FUNCTION_BLOCK FB_TP_LTIME (* standard timer function block (pulse) (LTIME) *)
  (* Standard: 61131-3; Classification: standard timer function block; Description: Copyright (c) 2011 TU Wien ACIN, Patrick Aigner, HR Agrartechnik GmbH This program and the accompanying materials are made available under the terms of the Eclipse Public License 2.0 which is available at https://www.eclipse.org/legal/epl-2.0/ SPDX-License-Identifier: EPL-2.0 Some portions generated by Gemini CLI *)
  (* Version 1.0, 2026-02-01, Franz Höpfinger, HR Agrartechnik GmbH, Copy over from FB_TP and made this Block *)
  PACKAGE iec61131::timers;
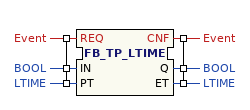
  EVENT_INPUT
    REQ WITH IN, PT; (* Service Request *)
  END_EVENT
  EVENT_OUTPUT
    CNF WITH Q, ET; (* Confirmation of Requested Service *)
  END_EVENT
  VAR_INPUT
    IN : BOOL; (* Input *)
    PT : LTIME; (* Pulse time *)
  END_VAR
  VAR_OUTPUT
    Q : BOOL; (* output *)
    ET : LTIME; (* elapse time *)
  END_VAR
  VAR
    MEM : BOOL; (* internal variable *)
    StartTime : LTIME; (* internal variable *)
  END_VAR
  EC_STATES
    REQ : REQ -> CNF;
  END_STATES
  ALGORITHM REQ IN ST:
VAR_TEMP
	SysTime : TIME;
END_VAR

SysTime := NOW_MONOTONIC();

IF IN AND NOT MEM THEN
	MEM := TRUE;

	IF NOT Q THEN
		Q := TRUE;
		ET := T#0s;
		StartTime := SysTime;
	END_IF;

ELSIF NOT IN THEN
	MEM := FALSE;
END_IF;

IF Q THEN
	ET := SysTime - StartTime;

	IF ET >= PT THEN
		Q := FALSE;
		ET := PT;
	END_IF;
END_IF;

IF NOT IN AND NOT Q THEN
	ET := T#0s;
END_IF;
  END_ALGORITHM
END_FUNCTION_BLOCK
